Fanuc KAREL source: kt00858.KL

-- PROVISIONAL review KL for V1013-1; original PC SHA256 7db11f5a503c37a99df30d48151a5a180c8efcd4a0f2e782c40117c0a705f4d5
-- Incomplete behavior may be omitted. Consult companion uncertainty JSON. Do not deploy.
PROGRAM KT00858
%NOLOCKGROUP
VAR
  R1 : REAL
  R2 : REAL
  OUT : INTEGER
BEGIN
  -- UNRESOLVED_PC offsets 5-16; opcodes 2E,23
  -- UNRESOLVED_PC offsets 21-32; opcodes 2E,23
  -- UNRESOLVED_PC offsets 37-48; opcodes 2E,23
  -- UNRESOLVED_PC offsets 53-64; opcodes 2E,23
  -- UNRESOLVED_PC offsets 69-84; opcodes 27,22,76,23
  -- UNRESOLVED_PC offsets 89-93; opcodes 7F
END KT00858
